(* CODESYS project TrabalhoFMS.project

Project tree, tasks and I/O mapping:
  Device : CODESYS Control Win V3, 3S - Smart Software Solutions GmbH, order no. 305021, version 3.5.11.30
    application Application
      libraries: Standard, * (System)
      task MainTask (cyclic, interval t#20ms, priority 1) calls PLC_PRG, LinhaFabricacao
      program PLC_PRG [SFC]
      program LinhaFabricacao [SFC]
      Symbols
*)

// Device/Application/PLC_PRG
PROGRAM PLC_PRG
VAR
	teste:BOOL;
	
END_VAR

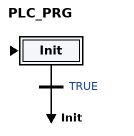
INITIAL_STEP Init:
END_STEP
TRANSITION FROM Init TO Init
    := TRUE;
END_TRANSITION

END_PROGRAM

// Device/Application/LinhaFabricacao
PROGRAM LinhaFabricacao
VAR
//saidas 
Conveyor6m1:BOOL;
ConveyorG1:BOOL;
Conveyor6m2:BOOL;
//entradas
SensorDifuso2:BOOL;

	Q1 AT %QX1.0: BOOL;
END_VAR

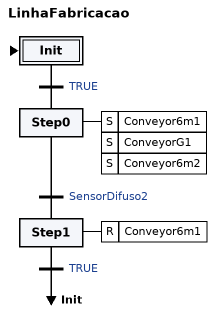
INITIAL_STEP Init:
END_STEP
TRANSITION FROM Init TO Step0
    := TRUE;
END_TRANSITION
STEP Step0:
    Conveyor6m1(S);
    ConveyorG1(S);
    Conveyor6m2(S);
END_STEP
TRANSITION FROM Step0 TO Step1
    := SensorDifuso2;
END_TRANSITION
STEP Step1:
    Conveyor6m1(R);
END_STEP
TRANSITION FROM Step1 TO Init
    := TRUE;
END_TRANSITION

END_PROGRAM
